{attribute 'qualified_only'}
VAR_GLOBAL
	globButtonYellow AT %I*: BOOL;
	globButtonBlue AT %I*: BOOL;
	globLightGreen AT %Q*: BOOL;
	globLightRed AT %Q*: BOOL;
END_VAR

(* stored: Version 1.1.0.1, ProductVersion 3.1.4022.12
   GVL GVL: Id {c8c933eb-708e-4875-8832-8c4bc0f55c82} *)
